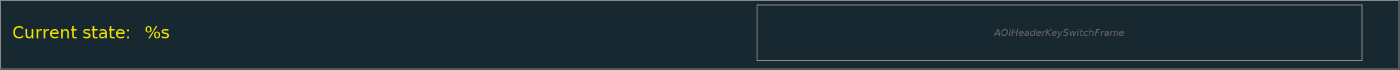
VISUALIZATION AOIHeaderFrame  // 1480x75
VAR_IN_OUT
	eMachineStateAutoFcqText 	: E_MachineCtrlStateAutoFcq;
	stDoorLock	 				: ST_VisuCtrlDoorLock;
END_VAR
    Label (10,15 150x40), "Current state:"
    Textfield (150,15 600x40), "%s", text list: 'TL_Fcq', text index: eMachineStateAutoFcqText
    Frame (800,5 640x60), invisible if: stDoorLock.bDoorLockInvisible
        shows AOIHeaderKeySwitchFrame()
END_VISUALIZATION

(* stored: Version 1.1.0.1, ProductVersion 3.1.4024.9
   Visu AOIHeaderFrame: Id {a477d5ae-c918-44c9-933c-56530a758c63} *)
